{attribute 'qualified_only'}
{attribute 'strict'}
TYPE E_WaterLevel :
(
	LOW := 1,
	MODERATE,
	HIGH
);
END_TYPE

(* stored: Version 1.1.0.1, ProductVersion 3.1.4024.16
   DUT E_WaterLevel: Id {8804dc95-49c3-4f7d-86b7-b47794d4770d} *)
